PROGRAM MAIN
VAR
	fbWeatherStation : FB_WeatherStation;
END_VAR

fbWeatherStation();

END_PROGRAM

(* stored: Version 1.1.0.1, ProductVersion 3.1.4024.12
   POU MAIN: Id {ffecc0be-3ece-405c-bd0b-1ec36ceb0d51}, SpecialFunc None *)
